FUNCTION_BLOCK FB_2In IMPLEMENTS  I_ConveyerSection
VAR_INPUT
END_VAR
VAR_OUTPUT
END_VAR
VAR
	stRack	: ST_2In;
	nStep	: UINT;
	bStart	: BOOL;
	_mDwnStrmHndShkIn	: BOOL;
	_mDwnStrmHndShkOut	: BOOL;
	_mUpStrmHndShkIn	: BOOL;
	_mUpStrmHndShkOut	: BOOL;
	_mId				: UINT;
	_mHMI				: ARRAY[0..15] OF BOOL;
	_mPosition			: INT;
END_VAR

Sequence();


PROPERTY DwnStrmHndShkIn : BOOL
SET
_mDwnStrmHndShkIn := DwnStrmHndShkIn;
END_SET
END_PROPERTY


PROPERTY DwnStrmHndShkOut : BOOL
GET
DwnStrmHndShkOut := _mDwnStrmHndShkOut;
END_GET
END_PROPERTY

{warning 'add property implementation'}
PROPERTY HMI : ARRAY [0..15] OF BOOL
GET
_mHMI[0] := stRack.ST_In1.Input1;
_mHMI[1] := stRack.ST_In1.Input2;
_mHMI[2] := stRack.ST_In1.Input3;
_mHMI[3] := stRack.ST_In1.Input4;
_mHMI[4] := stRack.ST_In1.Input5;
_mHMI[5] := stRack.ST_In1.Input6;
_mHMI[6] := stRack.ST_In1.Input7;
_mHMI[7] := stRack.ST_In1.Input8;
_mHMI[8] := stRack.ST_In2.Input1;
_mHMI[9] := stRack.ST_In2.Input2;
_mHMI[10] := stRack.ST_In2.Input3;
_mHMI[11] := stRack.ST_In2.Input4;
_mHMI[12] := stRack.ST_In2.Input5;
_mHMI[13] := stRack.ST_In2.Input6;
_mHMI[14] := stRack.ST_In2.Input7;
_mHMI[15] := stRack.ST_In2.Input8;
HMI := _mHMI;
END_GET
END_PROPERTY


PROPERTY Id : UINT
GET
Id := _mId;
END_GET
SET
_mId := Id;
END_SET
END_PROPERTY

{warning 'add property implementation'}
PROPERTY Pos : INT
GET
Pos := _mPosition;
END_GET
SET
_mPosition := Pos;
END_SET
END_PROPERTY


METHOD  Sequence : BOOL
IF _mDwnStrmHndShkIn THEN
	stRack.ST_In1.Input1 := TRUE;
	stRack.ST_In1.Input3 := TRUE;
	stRack.ST_In1.Input5 := TRUE;
	stRack.ST_In1.Input7 := TRUE;
END_IF

IF _mUpStrmHndShkIn THEN
	stRack.ST_In1.Input2 := TRUE;
	stRack.ST_In1.Input4 := TRUE;
	stRack.ST_In1.Input6 := TRUE;
	stRack.ST_In1.Input8 := TRUE;
END_IF


THIS^._mDwnStrmHndShkOut := THIS^._mUpStrmHndShkIn;
END_METHOD


METHOD startSequence : BOOL
bStart := TRUE;
END_METHOD


METHOD stopSequence : BOOL
bStart := FALSE;
nStep := 0;
THIS^._mDwnStrmHndShkOut := FALSE;
THIS^._mUpStrmHndShkOut := FALSE;
END_METHOD


PROPERTY UpStrmHndShkIn : BOOL
SET
_mUpStrmHndShkIn := UpStrmHndShkIn;
END_SET
END_PROPERTY


PROPERTY UpStrmHndShkOut : BOOL
GET
END_GET
END_PROPERTY

END_FUNCTION_BLOCK

(* stored: Version 1.1.0.1, ProductVersion 3.1.4024.6
   POU FB_2In: Id {d67345b7-1c05-4cf9-b4bc-90fce0145c40}, SpecialFunc None
   Property DwnStrmHndShkIn: Id {47ab43a8-d837-471e-aa72-62917e197adc}
   Set Set: Id {bf94a575-99b4-4558-8c95-8f6eb0862569}
   Property DwnStrmHndShkOut: Id {3df8f44e-35f6-460c-91fc-2de2666ba547}
   Get Get: Id {00fcd3c5-8ed9-4428-bb37-ca6c6484a22f}
   Property HMI: Id {ac877b1a-1aed-4d39-a6d3-06e7732da32e}
   Get Get: Id {2c00b052-6871-44c4-9b2b-a52817f0e016}
   Property Id: Id {17982008-f853-46a6-bbe3-1abdbed0dc6b}
   Get Get: Id {5df31b02-4085-4daf-bb80-1eeeee350b13}
   Set Set: Id {4a69abc8-d4cf-4944-bf8e-a4dfc0f5c42d}
   Property Pos: Id {834814ab-857d-4dd2-b419-59ece6851dfc}
   Get Get: Id {018eaa60-9dda-4e1c-bba5-585b961629e0}
   Set Set: Id {67f86bce-15ec-4d38-9fee-5169608991eb}
   Method Sequence: Id {54fe5422-9231-4ba7-9cc0-64105a92e1f7}
   Method startSequence: Id {ceafef28-e0e5-43e7-a1c7-36865ab1b258}
   Method stopSequence: Id {98efd0c5-f499-410c-988a-e62833f8dd60}
   Property UpStrmHndShkIn: Id {6cdf8a22-4fa3-4641-977f-d2d61616464c}
   Set Set: Id {7de5a219-ed6a-4f43-8abe-4aeb79b39526}
   Property UpStrmHndShkOut: Id {c52b1e40-3fd6-44bb-ad7f-fb1db1bc72a5}
   Get Get: Id {89a7b7f5-b6ba-40d6-81ab-41a4387d5083} *)
